{attribute 'linkalways'} 
{attribute 'no_explicit_call' := 'This FB is a CLASS and must be accessed using methods or properties'}
{attribute 'enable_dynamic_creation'}
FUNCTION_BLOCK FINAL MOD_INT EXTENDS Node
VAR
	in1 : _INT(0);
	in2 : _INT(0);
	out : _INT(0);
END_VAR

METHOD PUBLIC Clone : I_Node
VAR
	pNode : POINTER TO MOD_INT;
END_VAR
pNode := __NEW(MOD_INT);
Clone := pNode^;
END_METHOD

METHOD FB_init : BOOL
VAR_INPUT
	bInitRetains : BOOL; // if TRUE, the retain variables are initialized (warm start / cold start)
	bInCopyCode : BOOL;  // if TRUE, the instance afterwards gets moved into the copy code (online change)
END_VAR
AddInput('in1',THIS^.in1);
AddInput('in2',THIS^.in2);
AddOutput('out', THIS^.out);
END_METHOD

METHOD PROTECTED OnExecute
VAR
END_VAR
out.Value := in1.Value MOD in2.Value;
END_METHOD

END_FUNCTION_BLOCK

(* stored: Version 1.1.0.1, ProductVersion 3.1.4024.15
   POU MOD_INT: Id {09e0f794-aa4b-4e17-bf18-6e4095698a37}, SpecialFunc None
   Folder Constructor: Id {b857da9b-4506-45cd-b8ba-c1e215ba1aec}
   Method Clone: Id {b534e4d1-745c-4c9e-ac9d-c6e05702c661}
   Method FB_init: Id {22bcc4b5-2a90-4aa2-adce-ca0f5a69943e}
   Method OnExecute: Id {f7f8c2a4-e3eb-4e10-a306-de7bf24af3c2} *)
